FUNCTION_BLOCK FB_ModeVelo
VAR_INPUT
	bExecute:BOOL;
	bReset: BOOL;
	fVelSet:LREAL:=0;
	stStatus: ST_INDRADRIVE_AXIS_STATUS;
END_VAR
VAR_OUTPUT
	fSpeedSetpoint:LREAL:=0;
	bError: BOOL;
	nErrorId: UDINT;
	sErrorStr: STRING:=GVL_ErrorCodes.nErrorCodeOKStr;
END_VAR
VAR_IN_OUT
	stCommands: ST_INDRADRIVE_AXIS_COMMAND;
END_VAR

// Function: Constant velocity of target main  motor
// Control will be performed by the drive.
// Author: Anders Sandström 2018

stCommands.eMotionMode :=e_Motion_mode.eJogPositive;
stCommands.eOperationMode:=e_Operation_mode_no.eSecondaryOpMode2;
IF bExecute THEN
	fSpeedSetpoint:=fVelSet;
ELSE
	fSpeedSetpoint:=0;
END_IF
stCommands.fCommandVelocity:=0; // Other mode

END_FUNCTION_BLOCK

(* stored: Version 1.1.0.1, ProductVersion 3.1.4024.6
   POU FB_ModeVelo: Id {c95731c8-4fe5-4d11-ab47-46b5e16e76f1}, SpecialFunc None *)
